// TIA Portal V19 export
TYPE "C501_VAR_KLH_TYPIC"
   STRUCT
      OBS { ExternalAccessible := 'False'; ExternalVisible := 'False'; ExternalWritable := 'False'} : USInt;   // Observeerbaarheid
      VAR_STS_NORM { ExternalAccessible := 'False'; ExternalVisible := 'False'; ExternalWritable := 'False'} : USInt;   // Ja = Klep in normale positie Nee = Niet in normale positie
      VAR_BSC { ExternalAccessible := 'False'; ExternalVisible := 'False'; ExternalWritable := 'False'} : USInt;   // Ja = Brandblusinstallatie onbeschikbaar als niet in normaal Nee = Brandblusinstallatie wordt niet onbeschikbaar
   END_STRUCT;
END_TYPE
